// TwinCAT 3 PLC project ADSTestWithBool
// ProgramVersion: 3.1.4024.0
// libraries:
//   Tc2_Standard, * (Beckhoff Automation GmbH)
//   Tc2_System, * (Beckhoff Automation GmbH)
//   Tc3_Module, * (Beckhoff Automation GmbH)
// project tree:
//   / PlcTask.TcTTO (not stored)
//   POUs/ MAIN.TcPOU

// ---- POUs/MAIN.TcPOU
PROGRAM MAIN
VAR
	testBool			: BOOL := TRUE;
	testInt				: INT := 10;
	testString			: STRING(15)	:= 'Hello';
END_VAR

END_PROGRAM
